PROGRAM MAIN
VAR
	fbGetCurTaskIndex 	: GETCURTASKINDEX;
	f 					: INT := 0;
	g					: INT;
	
END_VAR


//Cycle count ja task-index kokeilu. alltwincat.com
//fbGetCurTaskIndex();
//	IF _TaskInfo[fbGetCurTaskIndex.index].FirstCycle THEN
//    // The code that you want to be executed at the first cycle
//	f :=1;				//first cycle kun on tosi, muutetaan ykköseksi. alustettu 0
//	g := g+1;			//ei alustettu lainkaan, lisätään g+1 tässä if-silmukassa (oletettavasti lisäisi 1ms välein +1 jos ei olis tätä silmukkaa)
//	GVL.h := GVL.h+1;	//GVL.h on persistent variable, lisää +1 jokasen restartin myötä
//	END_IF
	
//Liikennevalo
//MODE_SELECT();
//MODE_AUTO();
//MODE_MAN();
//VAIHE1();
//VAIHE2();
//VAIHE3();
//VAIHE4();
//VALO();

//extrat
//Lampotilailu();

END_PROGRAM

(* stored: Version 1.1.0.1, ProductVersion 3.1.4024.10
   POU MAIN: Id {44c959f8-a3ee-4249-ba7d-63d0439c89f3}, SpecialFunc None *)
